TYPE DATASTRUCT :
STRUCT
	p1:REAL;
	p2:REAL;
	p3:REAL;
	g:BOOL;
	h:BOOL;
END_STRUCT
END_TYPE

(* stored: Version 1.1.0.1, ProductVersion 3.1.0.38
   DUT DATASTRUCT: Id {b6461333-2eb5-47da-b98a-85380fcf24e3} *)
